// Home PLC
PROGRAM MAIN
VAR
	fbHome			: FB_MyHome;
	fbSimulation	: FB_Simulation;
END_VAR

fbHome.Execute();
//fbSimulation.Execute();

END_PROGRAM

(* stored: Version 1.1.0.1, ProductVersion 3.1.4024.12
   POU MAIN: Id {a6f55ad0-0d5e-4415-bd18-cbd370167f45}, SpecialFunc None *)
